// TIA Portal V17 export
// export: Created 2025-03-05T08:03:36.6878086Z, ExportSetting WithDefaults, DisplayName Totally Integrated Automation Portal, DisplayVersion V17 Update 8, DisplayName TIA Portal Openness, DisplayVersion V17 Update 8, DisplayName TIA Portal Version Control Interface, DisplayVersion V17, DisplayName SINAMICS Startdrive Advanced, DisplayVersion V17 SP2, DisplayName SINAMICS Startdrive G110M, G120, G120C, G120D, G120P, G115D, DisplayVersion V17 SP2, DisplayName SINAMICS Startdrive G130, G150, S120, S150, SINAMICS MV, S210, DisplayVersion V17 SP2, DisplayName STEP 7 Professional, DisplayVersion V17 Update 8, DisplayName SINUMERIK ONE STEP 7 Toolbox, DisplayVersion V17 Update 12, DisplayName SINUMERIK 840D sl STEP 7 Toolbox, DisplayVersion V17 Update 12, DisplayName STEP 7 Safety, DisplayVersion V17 Update 6, DisplayName WinCC Advanced, DisplayVersion V17 Update 8
DATA_BLOCK "DB1018_POWDER_NCU_SAFE_SIGNALS"   // DB1018, F_DB
{ S7_Optimized_Access := 'TRUE'; DB_Accessible_From_OPC_UA := 'FALSE' }
VERSION : 0.1
// stored: AutoNumber false, DBAccessibleFromOPCUA false, DBAccessibleFromWebserver true
   VAR
      E_STOP_OK_FROM_NCU : Bool;   // EMERGENCY STOP FROM MACHINE NCU
      SAFE_GATES_UNIT01_FROM_NCU : Bool;   // SAFETY GATES UNIT 01 CLOSED AND LOCKED FROM MACHINE NCU
      SAFE_GATES_UNIT02_FROM_NCU : Bool;   // SAFETY GATES UNIT 02 CLOSED AND LOCKED FROM MACHINE NCU
      POWER_ENABLE_UNIT_01_FROM_NCU : Bool;   // POWER ENABLE UNIT 01 FROM MACHINE NCU
      POWER_ENABLE_UNIT_02_FROM_NCU : Bool;   // POWER ENABLE UNIT 02 FROM MACHINE NCU
   END_VAR
BEGIN
END_DATA_BLOCK
